{attribute 'pack_mode' := '1'}
TYPE TProductionStats :
STRUCT
	rQualityRate			: REAL;
	rEfficiencyRate		: REAL;
	rAvailabilityRate		: REAL;
END_STRUCT
END_TYPE

(* stored: Version 1.1.0.1, ProductVersion 3.1.4022.12
   DUT TProductionStats: Id {332bd9a3-6f1d-4658-ba49-bee7115a4f37} *)
